(* CODESYS project T620X_HMI_CR1076_SP19p4.export

Project tree, tasks and I/O mapping:
  App_CODE_GEN/
    MAIN_CODE_GEN/
      App_CODE_GEN/
        Alarms/
          global variables GVL_Alarms
          program Alarms_Monitor_App [ST]
          program Alarms_Monitor_IO [ST]
        Diag_IO/
          program HMI_IO [FBD]: Init_Input_Links, Init_Output_Links, Update_Inputs, Update_Outputs
        Machine IO/
          Funcs/
            program Machine_Link_Inputs [ST]
            program Machine_Link_Inputs_Init [ST]
            program Machine_Link_Outputs [ST]
            program Machine_Link_Outputs_Init [ST]
            program Machine_Scale_Inputs [FBD]
          Structs/
            data type T620X_Radial_Inputs
            data type T620X_Radial_Outputs
    TEXT_LIST/
      text list AlarmGroup_App
      text list AlarmGroup_IO
      text list TextList_IO_Diag
*)

// App_CODE_GEN/MAIN_CODE_GEN/App_CODE_GEN/Machine IO/Structs/T620X_Radial_Inputs
TYPE T620X_Radial_Inputs :
STRUCT
// Machine_IO_Inputs_STRUCT_CODE_GEN_START

// generated (UTC): 2024-07-23 18:31:25.192393+00:00

ESTOP_OK:IpCom; // CHASSIS IN0100
DRUM_PRESSURE:IpCom; // CHASSIS IN0101
SPARE_IN0102:IpCom; // CHASSIS IN0102
SPARE_IN0103:IpCom; // CHASSIS IN0103
SPARE_IN0200:IpCom; // CHASSIS IN0200
SPARE_IN0201:IpCom; // CHASSIS IN0201
SPARE_IN0202:IpCom; // CHASSIS IN0202
SPARE_IN0203:IpCom; // CHASSIS IN0203
SPARE_IN0600:IpCom; // CHASSIS IN0600
SPARE_IN0601:IpCom; // CHASSIS IN0601
SPARE_IN0602:IpCom; // CHASSIS IN0602
SPARE_IN0603:IpCom; // CHASSIS IN0603
SPARE_IN0700:IpCom; // CHASSIS IN0700
RADIORHS_JACKLEGRAISE_REQ:IpCom; // CHASSIS IN0701
RHS_TROMMELDOORSW:IpCom; // CHASSIS IN0702
LHS_TROMMELDOORSW:IpCom; // CHASSIS IN0703
HYDOILTEMP_SW:IpCom; // CHASSIS IN0000
HYDOILLEVEL_SW:IpCom; // CHASSIS IN0001
THERMOSTAT:IpCom; // CHASSIS IN0002
RADIORHS_JACKLEGLOWER_REQ:IpCom; // CHASSIS IN0003
RADIOLHS_JACKLEGRAISE_REQ:IpCom; // CHASSIS IN0500
RADIOLHS_JACKLEGLOWER_REQ:IpCom; // CHASSIS IN0501
RADIOSIDECONVRAISEREQ:IpCom; // CHASSIS IN0502
RADIOSIDECONVLOWERREQ:IpCom; // CHASSIS IN0503
SPARE_IN0400:IpCom; // CHASSIS IN0400
FUELLEVEL_PERCENT:IpCom; // CHASSIS IN0401
UMBTRACKREQ:IpCom; // CHASSIS IN0900
UMBMACHINESTOP:IpCom; // CHASSIS IN0901
RTF_REQ:IpCom; // CHASSIS IN0300
RTR_REQ:IpCom; // CHASSIS IN0301
LTF_REQ:IpCom; // CHASSIS IN0800
LTR_REQ:IpCom; // CHASSIS IN0801


// Machine_IO_Inputs_STRUCT_CODE_GEN_STOP 

END_STRUCT
END_TYPE

// App_CODE_GEN/MAIN_CODE_GEN/App_CODE_GEN/Machine IO/Structs/T620X_Radial_Outputs
TYPE T620X_Radial_Outputs :
STRUCT
// Machine_IO_Outputs_STRUCT_CODE_GEN_START

// generated (UTC): 2024-07-23 18:31:25.208393+00:00

TAILCONVSPD_MA:OpCom; // CHASSIS.OUT0000
RHS_JACKLEGLOWER_OP:OpCom; // CHASSIS.OUT0001
SIDECONVSPD_MA:OpCom; // CHASSIS.OUT0002
LHS_JACKLEGRAISE_OP:OpCom; // CHASSIS.OUT0003
SIDETRANSFERSPD_MA:OpCom; // CHASSIS.OUT0004
LHS_JACKLEGLOWER_OP:OpCom; // CHASSIS.OUT0005
SETUPDUMPVALVE_OP:OpCom; // CHASSIS.OUT0006
COLLECTIONCONVSPD_MA:OpCom; // CHASSIS.OUT0007
COLLECTIONCONVON_OP:OpCom; // CHASSIS.OUT0008
SPARE_GROUP0:OpGrpCom; // CHASSIS.GROUP0
DRUMSPD_MA_RAMP_LIMIT:OpCom; // CHASSIS.OUT0100
TRACKINGMODE:OpCom; // CHASSIS.OUT0101
FEEDERSPD_MA:OpCom; // CHASSIS.OUT0102
CRANKENABLE:OpCom; // CHASSIS.OUT0103
DIVERTOILTOTRACK_OP:OpCom; // CHASSIS.OUT0104
RHS_JACKLEGRAISE_OP:OpCom; // CHASSIS.OUT0105
TAILCONVON_OP:OpCom; // CHASSIS.OUT0106
SIDECONVON_OP:OpCom; // CHASSIS.OUT0107
SIDETRANSFERON_OP:OpCom; // CHASSIS.OUT0108
SPARE_GROUP1:OpGrpCom; // CHASSIS.GROUP1
LEFTTRACKDIVERT_OP:OpCom; // CHASSIS.OUT0200
LTF_OP:OpCom; // CHASSIS.OUT0201
LTR_OP:OpCom; // CHASSIS.OUT0202
RIGHTTRACKDIVERT_OP:OpCom; // CHASSIS.OUT0203
RTF_OP:OpCom; // CHASSIS.OUT0204
RTR_OP:OpCom; // CHASSIS.OUT0205
DRUMONOFF_OP:OpCom; // CHASSIS.OUT0206
FEEDERONOFF_OP:OpCom; // CHASSIS.OUT0207
ECUENABLE:OpCom; // CHASSIS.OUT0208
SPARE_GROUP2:OpGrpCom; // CHASSIS.GROUP2
SPARE_OUT3000:OpCom; // CHASSIS.OUT3000
SPARE_OUT3001:OpCom; // CHASSIS.OUT3001


// Machine_IO_Outputs_STRUCT_CODE_GEN_STOP 	

END_STRUCT
END_TYPE

// App_CODE_GEN/MAIN_CODE_GEN/App_CODE_GEN/Alarms/GVL_Alarms
{attribute 'qualified_only'}
VAR_GLOBAL
// GVL_Alarms_Declare_CODE_GEN_START

// generated (UTC): 2024-07-23 18:31:25.263396+00:00

	EMERGENCY_STOP_COMMON: BOOL; // ID=101
	ETHERNET_PLC_COMMON_FAILURE: BOOL; // ID=102
	ETHERNET_CHASSIS_PLC_MISSING: BOOL; // ID=104
	ETHERNET_CHASSIS_PLC_ERROR_LT: BOOL; // ID=106
	ETHERNET_CHASSIS_PLC_ERROR_DIFF: BOOL; // ID=108
	ETHERNET_CHASSIS_PLC_ERROR_FROZEN: BOOL; // ID=110
	ETHERNET_CHASSIS_PLC_WARNING_DIFF: BOOL; // ID=112
	ETHERNET_CHASSIS_PLC_WARNING_FROZEN: BOOL; // ID=114
	Battery_Voltage_Warning: BOOL; // ID=118
	Hydraulic_Oil_Level_Low: BOOL; // ID=119
// GVL_Alarms_Declare_CODE_GEN_STOP
END_VAR

// App_CODE_GEN/MAIN_CODE_GEN/App_CODE_GEN/Alarms/Alarms_Monitor_App
PROGRAM Alarms_Monitor_App
VAR_INPUT
	LIST: REFERENCE TO SLL_LOGGER_MAIN_SRUCT;	
END_VAR
VAR
	App_Error_Group: SLL_LOGGER_ITEM_GROUP:=(ErrorApp:=1);	
	
// Alarms_Monitor_App_Declare_CODE_GEN_START

// generated (UTC): 2024-07-23 18:31:25.274396+00:00

	EMERGENCY_STOP_COMMON: SLL_AlarmBit;
	ETHERNET_PLC_COMMON_FAILURE: SLL_AlarmBit;
	ETHERNET_CHASSIS_PLC_MISSING: SLL_AlarmBit;
	ETHERNET_CHASSIS_PLC_ERROR_LT: SLL_AlarmBit;
	ETHERNET_CHASSIS_PLC_ERROR_DIFF: SLL_AlarmBit;
	ETHERNET_CHASSIS_PLC_ERROR_FROZEN: SLL_AlarmBit;
	ETHERNET_CHASSIS_PLC_WARNING_DIFF: SLL_AlarmBit;
	ETHERNET_CHASSIS_PLC_WARNING_FROZEN: SLL_AlarmBit;
	Battery_Voltage_Warning: SLL_AlarmBit;
	Hydraulic_Oil_Level_Low: SLL_AlarmBit;
	// Alarms_Monitor_App_Declare_CODE_GEN_STOP	
END_VAR


// Alarms_Monitor_App_STL_Body_CODE_GEN_START

// generated (UTC): 2024-07-23 18:31:25.284397+00:00

EMERGENCY_STOP_COMMON(LIST:=LIST,Bit_Input:=GVL_Alarms.EMERGENCY_STOP_COMMON,ID:=101,Add_Info:='',Group:=App_Error_Group,HushOption:=1);
ETHERNET_PLC_COMMON_FAILURE(LIST:=LIST,Bit_Input:=GVL_Alarms.ETHERNET_PLC_COMMON_FAILURE,ID:=102,Add_Info:='',Group:=App_Error_Group,HushOption:=0);
Battery_Voltage_Warning(LIST:=LIST,Bit_Input:=GVL_Alarms.Battery_Voltage_Warning,ID:=103,Add_Info:='',Group:=App_Error_Group,HushOption:=0);
Hydraulic_Oil_Level_Low(LIST:=LIST,Bit_Input:=GVL_Alarms.Hydraulic_Oil_Level_Low,ID:=104,Add_Info:='',Group:=App_Error_Group,HushOption:=0);

ETHERNET_CHASSIS_PLC_MISSING(LIST:=LIST,Bit_Input:=GVL_Alarms.ETHERNET_CHASSIS_PLC_MISSING,ID:=1100,Add_Info:='',Group:=App_Error_Group,HushOption:=0);
ETHERNET_CHASSIS_PLC_ERROR_LT(LIST:=LIST,Bit_Input:=GVL_Alarms.ETHERNET_CHASSIS_PLC_ERROR_LT,ID:=1101,Add_Info:='',Group:=App_Error_Group,HushOption:=0);
ETHERNET_CHASSIS_PLC_ERROR_DIFF(LIST:=LIST,Bit_Input:=GVL_Alarms.ETHERNET_CHASSIS_PLC_ERROR_DIFF,ID:=1102,Add_Info:='',Group:=App_Error_Group,HushOption:=0);
ETHERNET_CHASSIS_PLC_ERROR_FROZEN(LIST:=LIST,Bit_Input:=GVL_Alarms.ETHERNET_CHASSIS_PLC_ERROR_FROZEN,ID:=1103,Add_Info:='',Group:=App_Error_Group,HushOption:=0);
ETHERNET_CHASSIS_PLC_WARNING_DIFF(LIST:=LIST,Bit_Input:=GVL_Alarms.ETHERNET_CHASSIS_PLC_WARNING_DIFF,ID:=1104,Add_Info:='',Group:=App_Error_Group,HushOption:=0);
ETHERNET_CHASSIS_PLC_WARNING_FROZEN(LIST:=LIST,Bit_Input:=GVL_Alarms.ETHERNET_CHASSIS_PLC_WARNING_FROZEN,ID:=1105,Add_Info:='',Group:=App_Error_Group,HushOption:=0);




// Alarms_Monitor_App_STL_Body_CODE_GEN_STOP

END_PROGRAM

// App_CODE_GEN/MAIN_CODE_GEN/App_CODE_GEN/Alarms/Alarms_Monitor_IO
PROGRAM Alarms_Monitor_IO
VAR_INPUT
	LIST: REFERENCE TO SLL_LOGGER_MAIN_SRUCT;	
END_VAR
VAR
	IO_Error_Group: SLL_LOGGER_ITEM_GROUP:=(ErrorIO:=1);

// Alarms_Monitor_IO_Declare_CODE_GEN_START

// generated (UTC): 2024-07-23 18:31:25.297397+00:00

	ESTOPS_SAFETY_RELAY: SLL_AlarmBit;
	OVERRIDE_GENERAL_SWT: SLL_AlarmBit;
	FUNCTIONS_DEADMAN_CHASSIS_BTN: SLL_AlarmBit;
	CABIN_RAISE_CHASSIS_BTN: SLL_AlarmBit;
	CABIN_LOWER_CHASSIS_BTN: SLL_AlarmBit;
	JACKLEGS_DOWN_CHASSIS_BTN: SLL_AlarmBit;
	JACKLEGS_UP_CHASSIS_BTN: SLL_AlarmBit;
	ENGINE_START_CHASSIS_BTN: SLL_AlarmBit;
	HYDRAULICS_DC_PUMP_RUNNING_SIG: SLL_AlarmBit;
	JACKLEGS_STOWED_DOWN_PRESSURE_SWT: SLL_AlarmBit;
	JACKLEGS_STOWED_UP_PRESSURE_SWT: SLL_AlarmBit;
	MAINS_AC_MAINS_CONNECTED: SLL_AlarmBit;
	TRUCK_NEUTRAL_FROM_TRUCK : SLL_AlarmBit;
	SPARE_CHASSIS_IN0701: SLL_AlarmBit;
	CABIN_PART_RAISED_DIG: SLL_AlarmBit;
	SPARE_CHASSIS_IN0703: SLL_AlarmBit;
	CABIN_LOWER_LIMIT_DIG: SLL_AlarmBit;
	CABIN_FULLY_STOWED_DIG: SLL_AlarmBit;
	PTO_ACTIVE_SIG: SLL_AlarmBit;
	FUNCTIONS_CHASSIS_CABIN_CHANGE_OVER_SWT: SLL_AlarmBit;
	LIGHTS_SIDE_LIGHTS_DASH_SIG: SLL_AlarmBit;
	TRUCK_HANDBRAKE_APPLIED_SIGNAL: SLL_AlarmBit;
	ENGINE_RUNNING_SIGNAL: SLL_AlarmBit;
	TRUCK_REVERSE_FROM_TRUCK: SLL_AlarmBit;
	SPARE_CHASSIS_IN0400: SLL_AlarmBit;
	ENGINE_STOP_CHASSIS_BTN: SLL_AlarmBit;
	HYDRAULICS_OIL_LEVEL_RES: SLL_AlarmBit;
	SPARE_CHASSIS_IN0901: SLL_AlarmBit;
	SPARE_CHASSIS_IN0300: SLL_AlarmBit;
	SPARE_CHASSIS_IN0301: SLL_AlarmBit;
	JACKLEGS_CYCLINDER_100_BAR_PRESSURE_SWT: SLL_AlarmBit;
	JACKLEGS_CYCLINDER_150_BAR_PRESSURE_SWT: SLL_AlarmBit;
	ENGINE_STOP_COMMAND: SLL_AlarmBit;
	CHASSIS_SIREN: SLL_AlarmBit;
	SPARE_CHASSIS_OUT0002: SLL_AlarmBit;
	JACKLEGS_WARNING_BEACON: SLL_AlarmBit;
	HYDRAULICS_OIL_LEVEL_WARNING_LED: SLL_AlarmBit;
	SPARE_CHASSIS_OUT0005: SLL_AlarmBit;
	HYDRAULICS_MASTER_VALVE: SLL_AlarmBit;
	PTO_TOGGLE: SLL_AlarmBit;
	SPARE_CHASSIS_OUT0008: SLL_AlarmBit;
	CHASSIS_Supply_GROUP0: SLL_AlarmBit;
	SPARE_CHASSIS_OUT0100: SLL_AlarmBit;
	ENGINE_START_COMMAND: SLL_AlarmBit;
	SPARE_CHASSIS_OUT0102: SLL_AlarmBit;
	PLATFORM_TRAVERSE_LEFT_VALVE: SLL_AlarmBit;
	SPARE_CHASSIS_OUT0104: SLL_AlarmBit;
	CABIN_RAISE_COMMAND: SLL_AlarmBit;
	CABIN_LOWER_COMMAND: SLL_AlarmBit;
	JACKLEGS_UP_COMMAND: SLL_AlarmBit;
	JACKLEGS_DOWN_COMMAND: SLL_AlarmBit;
	CHASSIS_Supply_GROUP1: SLL_AlarmBit;
	HYDRAULICS_MASTER_LED_CAB: SLL_AlarmBit;
	OVERRIDE_DRIVE_INTERLOCK_ACTIVE_LED: SLL_AlarmBit;
	CABIN_FULLY_STOWED_LED: SLL_AlarmBit;
	JACKLEGS_STOWED_LED: SLL_AlarmBit;
	JACKLEGS_DOWN_LED: SLL_AlarmBit;
	CABIN_RAISED_LED: SLL_AlarmBit;
	PLATFORM_TRAVERSE_RIGHT_VALVE: SLL_AlarmBit;
	PLATFORM_RETRACT_COMMAND: SLL_AlarmBit;
	PLATFORM_EXTEND_COMMAND: SLL_AlarmBit;
	CHASSIS_Supply_GROUP2: SLL_AlarmBit;
	SPARE_CHASSIS_OUT3000: SLL_AlarmBit;
	SPARE_CHASSIS_OUT3001: SLL_AlarmBit;
	SPARE_CABIN_IN0100: SLL_AlarmBit;
	PLATFORM_EXTEND_BTN: SLL_AlarmBit;
	PLATFORM_RETRACT_BTN: SLL_AlarmBit;
	PLATFORM_SIDERAILS_LHS_SIDERAILS_STOWED_DIG: SLL_AlarmBit;
	PLATFORM_SIDERAILS_RHS_SIDERAILS_STOWED_DIG: SLL_AlarmBit;
	PLATFORM_TRAVERSE_STOWED_DIG: SLL_AlarmBit;
	SPARE_CABIN_IN0202: SLL_AlarmBit;
	PLATFORM_LEUZE_SENSORS_LEFT_SENSOR_DIG: SLL_AlarmBit;
	PLATFORM_LEUZE_SENSORS_RIGHT_SENSOR_DIG: SLL_AlarmBit;
	PLATFORM_FULLY_STOWED_DIG: SLL_AlarmBit;
	PLATFORM_PART_STOWED_DIG: SLL_AlarmBit;
	DOORS_REAR_DOOR_CLOSED_SIG: SLL_AlarmBit;
	PLATFORM_SAFETY_GATES_LHS_EDGE_SENSOR: SLL_AlarmBit;
	SPARE_CABIN_IN0701: SLL_AlarmBit;
	SPARE_CABIN_IN0702: SLL_AlarmBit;
	PLATFORM_SAFETY_GATES_RHS_EDGE_SENSOR: SLL_AlarmBit;
	SPARE_CABIN_IN0000: SLL_AlarmBit;
	PLATFORM_SAFETY_GATES_LHS_GATE_CLOSED_SIGNAL: SLL_AlarmBit;
	PLATFORM_SAFETY_GATES_RHS_GATE_CLOSED_SIGNAL: SLL_AlarmBit;
	SPARE_CABIN_IN0003: SLL_AlarmBit;
	CAS_RESET_SWT: SLL_AlarmBit;
	CAS_TORTOISE_SWT: SLL_AlarmBit;
	CAS_ENABLE_ON_OFF_SWT: SLL_AlarmBit;
	SPARE_CABIN_IN0503: SLL_AlarmBit;
	PLATFORM_SAFETY_EDGE_SAFETY_BUMPER_RES_ANA: SLL_AlarmBit;
	SPARE_CABIN_IN0401: SLL_AlarmBit;
	PLATFORM_TRAVERSE_LEFT_BTN: SLL_AlarmBit;
	PLATFORM_TRAVERSE_RIGHT_BTN: SLL_AlarmBit;
	DOORS_SIDE_DOOR_CLOSED_SIG: SLL_AlarmBit;
	FUNCTIONS_DEADMAN_CABIN_BTN: SLL_AlarmBit;
	SPARE_CABIN_IN0800: SLL_AlarmBit;
	SPARE_CABIN_IN0801: SLL_AlarmBit;
	PLATFORM_SIDERAILS_SIDERAILS_STOWED_LED: SLL_AlarmBit;
	PLATFORM_SAFETY_GATES_UNLOCK_1: SLL_AlarmBit;
	TRUCK_FORCE_NEUTRAL: SLL_AlarmBit;
	PLATFORM_SAFETY_GATES_UNLOCK_2: SLL_AlarmBit;
	CAS_LOCKOUT_LED: SLL_AlarmBit;
	PLATFORM_EXTENDED_LED: SLL_AlarmBit;
	PLATFORM_RETRACTED_LED: SLL_AlarmBit;
	CAS_TORTOISE_MODE_LED: SLL_AlarmBit;
	CAS_DRIVERS_BUZZER: SLL_AlarmBit;
	CABIN_Supply_GROUP0: SLL_AlarmBit;
	DOORS_ALLOW_SIDE_DOOR: SLL_AlarmBit;
	DOORS_ALLOW_REAR_DOOR: SLL_AlarmBit;
	SPARE_CABIN_OUT0102: SLL_AlarmBit;
	SPARE_CABIN_OUT0103: SLL_AlarmBit;
	SPARE_CABIN_OUT0104: SLL_AlarmBit;
	SPARE_CABIN_OUT0105: SLL_AlarmBit;
	SPARE_CABIN_OUT0106: SLL_AlarmBit;
	SPARE_CABIN_OUT0107: SLL_AlarmBit;
	SPARE_CABIN_OUT0108: SLL_AlarmBit;
	CABIN_Supply_GROUP1: SLL_AlarmBit;
	SPARE_CABIN_OUT0200: SLL_AlarmBit;
	LIGHTS_LEFT_SIDE_LIGHTS: SLL_AlarmBit;
	CAS_GREEN_BEACON: SLL_AlarmBit;
	FUNCTIONS_DEADMAN_CABIN_BTN_LED: SLL_AlarmBit;
	SPARE_CABIN_OUT0204: SLL_AlarmBit;
	SPARE_CABIN_OUT0205: SLL_AlarmBit;
	LIGHTS_SIDE_RLY: SLL_AlarmBit;
	SPARE_CABIN_OUT0207: SLL_AlarmBit;
	SPARE_CABIN_OUT0208: SLL_AlarmBit;
	CABIN_Supply_GROUP2: SLL_AlarmBit;
	SPARE_CABIN_OUT3000: SLL_AlarmBit;
	SPARE_CABIN_OUT3001: SLL_AlarmBit;
	// Alarms_Monitor_IO_Declare_CODE_GEN_STOP	
END_VAR


// Alarms_Monitor_IO_STL_Body_CODE_GEN_START

// generated (UTC): 2024-07-23 18:31:25.307398+00:00

// Alarms_Monitor_IO_STL_Body_CODE_GEN_STOP

END_PROGRAM

// App_CODE_GEN/MAIN_CODE_GEN/App_CODE_GEN/Diag_IO/HMI_IO
PROGRAM HMI_IO
VAR
	Init_Link_Inputs: BOOL:=TRUE;
	Init_Link_Outputs: BOOL:=TRUE;
	CHASSIS: HMI_PLC_CR0709_IO;	
	Outputs_EnableAutoMan:BOOL:=TRUE;// AW TEMP 02-03-2024
	Wait_For_UDP_TON: TON;
END_VAR

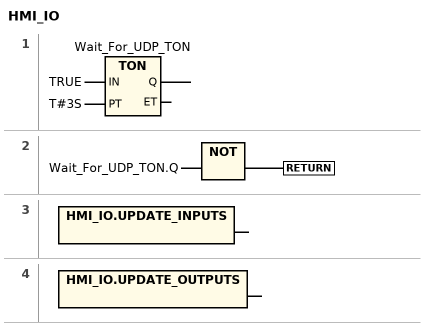
// NETWORK 1
Wait_For_UDP_TON(IN := TRUE, PT := T#3S); // TON

// NETWORK 2
IF NOT Wait_For_UDP_TON.Q THEN RETURN; END_IF

// NETWORK 3
HMI_IO.UPDATE_INPUTS();

// NETWORK 4
HMI_IO.UPDATE_OUTPUTS();

METHOD Init_Input_Links
VAR
END_VAR

// HMI_IO_Init_Input_Links_CODE_GEN_START

// generated (UTC): 2024-07-23 18:31:25.317398+00:00
CHASSIS.IN0100.Init(Machine_IO.Inputs.ESTOP_OK);
CHASSIS.IN0101.Init(Machine_IO.Inputs.DRUM_PRESSURE);
CHASSIS.IN0102.Init(Machine_IO.Inputs.SPARE_IN0102);
CHASSIS.IN0103.Init(Machine_IO.Inputs.SPARE_IN0103);
CHASSIS.IN0200.Init(Machine_IO.Inputs.SPARE_IN0200);
CHASSIS.IN0201.Init(Machine_IO.Inputs.SPARE_IN0201);
CHASSIS.IN0202.Init(Machine_IO.Inputs.SPARE_IN0202);
CHASSIS.IN0203.Init(Machine_IO.Inputs.SPARE_IN0203);
CHASSIS.IN0600.Init(Machine_IO.Inputs.SPARE_IN0600);
CHASSIS.IN0601.Init(Machine_IO.Inputs.SPARE_IN0601);
CHASSIS.IN0602.Init(Machine_IO.Inputs.SPARE_IN0602);
CHASSIS.IN0603.Init(Machine_IO.Inputs.SPARE_IN0603);
CHASSIS.IN0700.Init(Machine_IO.Inputs.SPARE_IN0700);
CHASSIS.IN0701.Init(Machine_IO.Inputs.RADIORHS_JACKLEGRAISE_REQ);
CHASSIS.IN0702.Init(Machine_IO.Inputs.RHS_TROMMELDOORSW);
CHASSIS.IN0703.Init(Machine_IO.Inputs.LHS_TROMMELDOORSW);
CHASSIS.IN0000.Init(Machine_IO.Inputs.HYDOILTEMP_SW);
CHASSIS.IN0001.Init(Machine_IO.Inputs.HYDOILLEVEL_SW);
CHASSIS.IN0002.Init(Machine_IO.Inputs.THERMOSTAT);
CHASSIS.IN0003.Init(Machine_IO.Inputs.RADIORHS_JACKLEGLOWER_REQ);
CHASSIS.IN0500.Init(Machine_IO.Inputs.RADIOLHS_JACKLEGRAISE_REQ);
CHASSIS.IN0501.Init(Machine_IO.Inputs.RADIOLHS_JACKLEGLOWER_REQ);
CHASSIS.IN0502.Init(Machine_IO.Inputs.RADIOSIDECONVRAISEREQ);
CHASSIS.IN0503.Init(Machine_IO.Inputs.RADIOSIDECONVLOWERREQ);
CHASSIS.IN0400.Init(Machine_IO.Inputs.SPARE_IN0400);
CHASSIS.IN0401.Init(Machine_IO.Inputs.FUELLEVEL_PERCENT);
CHASSIS.IN0900.Init(Machine_IO.Inputs.UMBTRACKREQ);
CHASSIS.IN0901.Init(Machine_IO.Inputs.UMBMACHINESTOP);
CHASSIS.IN0300.Init(Machine_IO.Inputs.RTF_REQ);
CHASSIS.IN0301.Init(Machine_IO.Inputs.RTR_REQ);
CHASSIS.IN0800.Init(Machine_IO.Inputs.LTF_REQ);
CHASSIS.IN0801.Init(Machine_IO.Inputs.LTR_REQ);

// HMI_IO_Init_Input_Links_CODE_GEN_STOP
END_METHOD

METHOD Init_Output_Links
VAR
END_VAR

// HMI_IO_Init_Output_Links_CODE_GEN_START

// generated (UTC): 2024-07-23 18:31:25.327399+00:00
CHASSIS.OUT0000.Init(Machine_IO.Outputs.TAILCONVSPD_MA);
CHASSIS.OUT0001.Init(Machine_IO.Outputs.RHS_JACKLEGLOWER_OP);
CHASSIS.OUT0002.Init(Machine_IO.Outputs.SIDECONVSPD_MA);
CHASSIS.OUT0003.Init(Machine_IO.Outputs.LHS_JACKLEGRAISE_OP);
CHASSIS.OUT0004.Init(Machine_IO.Outputs.SIDETRANSFERSPD_MA);
CHASSIS.OUT0005.Init(Machine_IO.Outputs.LHS_JACKLEGLOWER_OP);
CHASSIS.OUT0006.Init(Machine_IO.Outputs.SETUPDUMPVALVE_OP);
CHASSIS.OUT0007.Init(Machine_IO.Outputs.COLLECTIONCONVSPD_MA);
CHASSIS.OUT0008.Init(Machine_IO.Outputs.COLLECTIONCONVON_OP);
CHASSIS.GROUP0.Init(Machine_IO.Outputs.SPARE_GROUP0);
CHASSIS.OUT0100.Init(Machine_IO.Outputs.DRUMSPD_MA_RAMP_LIMIT);
CHASSIS.OUT0101.Init(Machine_IO.Outputs.TRACKINGMODE);
CHASSIS.OUT0102.Init(Machine_IO.Outputs.FEEDERSPD_MA);
CHASSIS.OUT0103.Init(Machine_IO.Outputs.CRANKENABLE);
CHASSIS.OUT0104.Init(Machine_IO.Outputs.DIVERTOILTOTRACK_OP);
CHASSIS.OUT0105.Init(Machine_IO.Outputs.RHS_JACKLEGRAISE_OP);
CHASSIS.OUT0106.Init(Machine_IO.Outputs.TAILCONVON_OP);
CHASSIS.OUT0107.Init(Machine_IO.Outputs.SIDECONVON_OP);
CHASSIS.OUT0108.Init(Machine_IO.Outputs.SIDETRANSFERON_OP);
CHASSIS.GROUP1.Init(Machine_IO.Outputs.SPARE_GROUP1);
CHASSIS.OUT0200.Init(Machine_IO.Outputs.LEFTTRACKDIVERT_OP);
CHASSIS.OUT0201.Init(Machine_IO.Outputs.LTF_OP);
CHASSIS.OUT0202.Init(Machine_IO.Outputs.LTR_OP);
CHASSIS.OUT0203.Init(Machine_IO.Outputs.RIGHTTRACKDIVERT_OP);
CHASSIS.OUT0204.Init(Machine_IO.Outputs.RTF_OP);
CHASSIS.OUT0205.Init(Machine_IO.Outputs.RTR_OP);
CHASSIS.OUT0206.Init(Machine_IO.Outputs.DRUMONOFF_OP);
CHASSIS.OUT0207.Init(Machine_IO.Outputs.FEEDERONOFF_OP);
CHASSIS.OUT0208.Init(Machine_IO.Outputs.ECUENABLE);
CHASSIS.GROUP2.Init(Machine_IO.Outputs.SPARE_GROUP2);
CHASSIS.OUT3000.Init(Machine_IO.Outputs.SPARE_OUT3000);
CHASSIS.OUT3001.Init(Machine_IO.Outputs.SPARE_OUT3001);

// HMI_IO_Init_Output_Links_CODE_GEN_STOP
END_METHOD

METHOD Update_Inputs
VAR	
END_VAR
IF Init_Link_Inputs THEN
	Init_Input_Links();
END_IF
Init_Link_Inputs:=FALSE;

// HMI_IO_Update_Inputs_CODE_GEN_START

// generated (UTC): 2024-07-23 18:31:25.338400+00:00

CHASSIS.IN0100();
CHASSIS.IN0101();
CHASSIS.IN0102();
CHASSIS.IN0103();
CHASSIS.IN0200();
CHASSIS.IN0201();
CHASSIS.IN0202();
CHASSIS.IN0203();
CHASSIS.IN0600();
CHASSIS.IN0601();
CHASSIS.IN0602();
CHASSIS.IN0603();
CHASSIS.IN0700();
CHASSIS.IN0701();
CHASSIS.IN0702();
CHASSIS.IN0703();
CHASSIS.IN0000();
CHASSIS.IN0001();
CHASSIS.IN0002();
CHASSIS.IN0003();
CHASSIS.IN0500();
CHASSIS.IN0501();
CHASSIS.IN0502();
CHASSIS.IN0503();
CHASSIS.IN0400();
CHASSIS.IN0401();
CHASSIS.IN0900();
CHASSIS.IN0901();
CHASSIS.IN0300();
CHASSIS.IN0301();
CHASSIS.IN0800();
CHASSIS.IN0801();
// HMI_IO_Update_Inputs_CODE_GEN_STOP
END_METHOD

METHOD Update_Outputs
VAR
END_VAR
IF Init_Link_Outputs THEN
	Init_Output_Links();
END_IF
Init_Link_Outputs:=FALSE;

// HMI_IO_Update_Outputs_CODE_GEN_START

// generated (UTC): 2024-07-23 18:31:25.349399+00:00

CHASSIS.OUT0000();
CHASSIS.OUT0001();
CHASSIS.OUT0002();
CHASSIS.OUT0003();
CHASSIS.OUT0004();
CHASSIS.OUT0005();
CHASSIS.OUT0006();
CHASSIS.OUT0007();
CHASSIS.OUT0008();
CHASSIS.GROUP0();
CHASSIS.OUT0100();
CHASSIS.OUT0101();
CHASSIS.OUT0102();
CHASSIS.OUT0103();
CHASSIS.OUT0104();
CHASSIS.OUT0105();
CHASSIS.OUT0106();
CHASSIS.OUT0107();
CHASSIS.OUT0108();
CHASSIS.GROUP1();
CHASSIS.OUT0200();
CHASSIS.OUT0201();
CHASSIS.OUT0202();
CHASSIS.OUT0203();
CHASSIS.OUT0204();
CHASSIS.OUT0205();
CHASSIS.OUT0206();
CHASSIS.OUT0207();
CHASSIS.OUT0208();
CHASSIS.GROUP2();
CHASSIS.OUT3000();
CHASSIS.OUT3001();
// HMI_IO_Update_Outputs_CODE_GEN_STOP
END_METHOD

END_PROGRAM

// App_CODE_GEN/MAIN_CODE_GEN/App_CODE_GEN/Machine IO/Funcs/Machine_Link_Inputs
PROGRAM Machine_Link_Inputs
VAR_INPUT
	ENA:BOOL;
END_VAR

VAR
	INIT_ONCE:BOOL:=TRUE;
	Init_Input_Links:BOOL :=TRUE;
END_VAR

IF Init_Input_Links THEN
	Machine_Link_Inputs_Init();	
	Init_Input_Links:=FALSE;
END_IF

// Machine_Link_Inputs_Main_CODE_GEN_START

// generated (UTC): 2024-07-23 18:31:25.048386+00:00

Machine_IO.Inputs.ESTOP_OK(); // CR0709.IN0100
Machine_IO.Inputs.DRUM_PRESSURE(); // CR0709.IN0101
Machine_IO.Inputs.SPARE_IN0102(); // CR0709.IN0102
Machine_IO.Inputs.SPARE_IN0103(); // CR0709.IN0103
Machine_IO.Inputs.SPARE_IN0200(); // CR0709.IN0200
Machine_IO.Inputs.SPARE_IN0201(); // CR0709.IN0201
Machine_IO.Inputs.SPARE_IN0202(); // CR0709.IN0202
Machine_IO.Inputs.SPARE_IN0203(); // CR0709.IN0203
Machine_IO.Inputs.SPARE_IN0600(); // CR0709.IN0600
Machine_IO.Inputs.SPARE_IN0601(); // CR0709.IN0601
Machine_IO.Inputs.SPARE_IN0602(); // CR0709.IN0602
Machine_IO.Inputs.SPARE_IN0603(); // CR0709.IN0603
Machine_IO.Inputs.SPARE_IN0700(); // CR0709.IN0700
Machine_IO.Inputs.RADIORHS_JACKLEGRAISE_REQ(); // CR0709.IN0701
Machine_IO.Inputs.RHS_TROMMELDOORSW(); // CR0709.IN0702
Machine_IO.Inputs.LHS_TROMMELDOORSW(); // CR0709.IN0703
Machine_IO.Inputs.HYDOILTEMP_SW(); // CR0709.IN0000
Machine_IO.Inputs.HYDOILLEVEL_SW(); // CR0709.IN0001
Machine_IO.Inputs.THERMOSTAT(); // CR0709.IN0002
Machine_IO.Inputs.RADIORHS_JACKLEGLOWER_REQ(); // CR0709.IN0003
Machine_IO.Inputs.RADIOLHS_JACKLEGRAISE_REQ(); // CR0709.IN0500
Machine_IO.Inputs.RADIOLHS_JACKLEGLOWER_REQ(); // CR0709.IN0501
Machine_IO.Inputs.RADIOSIDECONVRAISEREQ(); // CR0709.IN0502
Machine_IO.Inputs.RADIOSIDECONVLOWERREQ(); // CR0709.IN0503
Machine_IO.Inputs.SPARE_IN0400(); // CR0709.IN0400
Machine_IO.Inputs.FUELLEVEL_PERCENT(); // CR0709.IN0401
Machine_IO.Inputs.UMBTRACKREQ(); // CR0709.IN0900
Machine_IO.Inputs.UMBMACHINESTOP(); // CR0709.IN0901
Machine_IO.Inputs.RTF_REQ(); // CR0709.IN0300
Machine_IO.Inputs.RTR_REQ(); // CR0709.IN0301
Machine_IO.Inputs.LTF_REQ(); // CR0709.IN0800
Machine_IO.Inputs.LTR_REQ(); // CR0709.IN0801


// Machine_Link_Inputs_Main_CODE_GEN_STOP

END_PROGRAM

// App_CODE_GEN/MAIN_CODE_GEN/App_CODE_GEN/Machine IO/Funcs/Machine_Link_Inputs_Init
PROGRAM Machine_Link_Inputs_Init
VAR
END_VAR


// Machine_Link_Inputs_Init_CODE_GEN_START

// generated (UTC): 2024-07-23 18:31:25.086388+00:00
Machine_IO.Inputs.ESTOP_OK.Init('CHASSIS','ESTOP_OK','IN0100','a63',NVL_IO_CHASSIS.All_Inputs.IN0100,Machine_IO.Node_CHASSIS);
Machine_IO.Inputs.DRUM_PRESSURE.Init('CHASSIS','DRUM_PRESSURE','IN0101','a64',NVL_IO_CHASSIS.All_Inputs.IN0101,Machine_IO.Node_CHASSIS);
Machine_IO.Inputs.SPARE_IN0102.Init('CHASSIS','SPARE_IN0102','IN0102','a65',NVL_IO_CHASSIS.All_Inputs.IN0102,Machine_IO.Node_CHASSIS);
Machine_IO.Inputs.SPARE_IN0103.Init('CHASSIS','SPARE_IN0103','IN0103','a66',NVL_IO_CHASSIS.All_Inputs.IN0103,Machine_IO.Node_CHASSIS);
Machine_IO.Inputs.SPARE_IN0200.Init('CHASSIS','SPARE_IN0200','IN0200','a67',NVL_IO_CHASSIS.All_Inputs.IN0200,Machine_IO.Node_CHASSIS);
Machine_IO.Inputs.SPARE_IN0201.Init('CHASSIS','SPARE_IN0201','IN0201','a68',NVL_IO_CHASSIS.All_Inputs.IN0201,Machine_IO.Node_CHASSIS);
Machine_IO.Inputs.SPARE_IN0202.Init('CHASSIS','SPARE_IN0202','IN0202','a69',NVL_IO_CHASSIS.All_Inputs.IN0202,Machine_IO.Node_CHASSIS);
Machine_IO.Inputs.SPARE_IN0203.Init('CHASSIS','SPARE_IN0203','IN0203','a70',NVL_IO_CHASSIS.All_Inputs.IN0203,Machine_IO.Node_CHASSIS);
Machine_IO.Inputs.SPARE_IN0600.Init('CHASSIS','SPARE_IN0600','IN0600','a55',NVL_IO_CHASSIS.All_Inputs.IN0600,Machine_IO.Node_CHASSIS);
Machine_IO.Inputs.SPARE_IN0601.Init('CHASSIS','SPARE_IN0601','IN0601','a56',NVL_IO_CHASSIS.All_Inputs.IN0601,Machine_IO.Node_CHASSIS);
Machine_IO.Inputs.SPARE_IN0602.Init('CHASSIS','SPARE_IN0602','IN0602','a57',NVL_IO_CHASSIS.All_Inputs.IN0602,Machine_IO.Node_CHASSIS);
Machine_IO.Inputs.SPARE_IN0603.Init('CHASSIS','SPARE_IN0603','IN0603','a58',NVL_IO_CHASSIS.All_Inputs.IN0603,Machine_IO.Node_CHASSIS);
Machine_IO.Inputs.SPARE_IN0700.Init('CHASSIS','SPARE_IN0700','IN0700','a59',NVL_IO_CHASSIS.All_Inputs.IN0700,Machine_IO.Node_CHASSIS);
Machine_IO.Inputs.RADIORHS_JACKLEGRAISE_REQ.Init('CHASSIS','RADIORHS_JACKLEGRAISE_REQ','IN0701','a60',NVL_IO_CHASSIS.All_Inputs.IN0701,Machine_IO.Node_CHASSIS);
Machine_IO.Inputs.RHS_TROMMELDOORSW.Init('CHASSIS','RHS_TROMMELDOORSW','IN0702','a61',NVL_IO_CHASSIS.All_Inputs.IN0702,Machine_IO.Node_CHASSIS);
Machine_IO.Inputs.LHS_TROMMELDOORSW.Init('CHASSIS','LHS_TROMMELDOORSW','IN0703','a62',NVL_IO_CHASSIS.All_Inputs.IN0703,Machine_IO.Node_CHASSIS);
Machine_IO.Inputs.HYDOILTEMP_SW.Init('CHASSIS','HYDOILTEMP_SW','IN0000','a25',NVL_IO_CHASSIS.All_Inputs.IN0000,Machine_IO.Node_CHASSIS);
Machine_IO.Inputs.HYDOILLEVEL_SW.Init('CHASSIS','HYDOILLEVEL_SW','IN0001','a26',NVL_IO_CHASSIS.All_Inputs.IN0001,Machine_IO.Node_CHASSIS);
Machine_IO.Inputs.THERMOSTAT.Init('CHASSIS','THERMOSTAT','IN0002','a27',NVL_IO_CHASSIS.All_Inputs.IN0002,Machine_IO.Node_CHASSIS);
Machine_IO.Inputs.RADIORHS_JACKLEGLOWER_REQ.Init('CHASSIS','RADIORHS_JACKLEGLOWER_REQ','IN0003','a28',NVL_IO_CHASSIS.All_Inputs.IN0003,Machine_IO.Node_CHASSIS);
Machine_IO.Inputs.RADIOLHS_JACKLEGRAISE_REQ.Init('CHASSIS','RADIOLHS_JACKLEGRAISE_REQ','IN0500','a40',NVL_IO_CHASSIS.All_Inputs.IN0500,Machine_IO.Node_CHASSIS);
Machine_IO.Inputs.RADIOLHS_JACKLEGLOWER_REQ.Init('CHASSIS','RADIOLHS_JACKLEGLOWER_REQ','IN0501','a41',NVL_IO_CHASSIS.All_Inputs.IN0501,Machine_IO.Node_CHASSIS);
Machine_IO.Inputs.RADIOSIDECONVRAISEREQ.Init('CHASSIS','RADIOSIDECONVRAISEREQ','IN0502','a42',NVL_IO_CHASSIS.All_Inputs.IN0502,Machine_IO.Node_CHASSIS);
Machine_IO.Inputs.RADIOSIDECONVLOWERREQ.Init('CHASSIS','RADIOSIDECONVLOWERREQ','IN0503','a43',NVL_IO_CHASSIS.All_Inputs.IN0503,Machine_IO.Node_CHASSIS);
Machine_IO.Inputs.SPARE_IN0400.Init('CHASSIS','SPARE_IN0400','IN0400','a46',NVL_IO_CHASSIS.All_Inputs.IN0400,Machine_IO.Node_CHASSIS);
Machine_IO.Inputs.FUELLEVEL_PERCENT.Init('CHASSIS','FUELLEVEL_PERCENT','IN0401','a47',NVL_IO_CHASSIS.All_Inputs.IN0401,Machine_IO.Node_CHASSIS);
Machine_IO.Inputs.UMBTRACKREQ.Init('CHASSIS','UMBTRACKREQ','IN0900','a38',NVL_IO_CHASSIS.All_Inputs.IN0900,Machine_IO.Node_CHASSIS);
Machine_IO.Inputs.UMBMACHINESTOP.Init('CHASSIS','UMBMACHINESTOP','IN0901','a39',NVL_IO_CHASSIS.All_Inputs.IN0901,Machine_IO.Node_CHASSIS);
Machine_IO.Inputs.RTF_REQ.Init('CHASSIS','RTF_REQ','IN0300','a44',NVL_IO_CHASSIS.All_Inputs.IN0300,Machine_IO.Node_CHASSIS);
Machine_IO.Inputs.RTR_REQ.Init('CHASSIS','RTR_REQ','IN0301','a45',NVL_IO_CHASSIS.All_Inputs.IN0301,Machine_IO.Node_CHASSIS);
Machine_IO.Inputs.LTF_REQ.Init('CHASSIS','LTF_REQ','IN0800','a36',NVL_IO_CHASSIS.All_Inputs.IN0800,Machine_IO.Node_CHASSIS);
Machine_IO.Inputs.LTR_REQ.Init('CHASSIS','LTR_REQ','IN0801','a37',NVL_IO_CHASSIS.All_Inputs.IN0801,Machine_IO.Node_CHASSIS);


// Machine_Link_Inputs_Init_CODE_GEN_STOP

END_PROGRAM

// App_CODE_GEN/MAIN_CODE_GEN/App_CODE_GEN/Machine IO/Funcs/Machine_Link_Outputs
PROGRAM Machine_Link_Outputs
VAR_INPUT
	ENA:BOOL;
END_VAR
VAR
	Init_Output_Links: BOOL := TRUE;
END_VAR

IF ENA = FALSE THEN
	RETURN;
END_IF

IF Init_Output_Links THEN
	Machine_Link_Outputs_Init();
	Init_Output_Links:=FALSE;
END_IF

// Machine_Link_Outputs_Main_CODE_GEN_START

// generated (UTC): 2024-07-23 18:31:25.127390+00:00
Machine_IO.Outputs.TAILCONVSPD_MA(); // CR0709.OUT0000
Machine_IO.Outputs.RHS_JACKLEGLOWER_OP(); // CR0709.OUT0001
Machine_IO.Outputs.SIDECONVSPD_MA(); // CR0709.OUT0002
Machine_IO.Outputs.LHS_JACKLEGRAISE_OP(); // CR0709.OUT0003
Machine_IO.Outputs.SIDETRANSFERSPD_MA(); // CR0709.OUT0004
Machine_IO.Outputs.LHS_JACKLEGLOWER_OP(); // CR0709.OUT0005
Machine_IO.Outputs.SETUPDUMPVALVE_OP(); // CR0709.OUT0006
Machine_IO.Outputs.COLLECTIONCONVSPD_MA(); // CR0709.OUT0007
Machine_IO.Outputs.COLLECTIONCONVON_OP(); // CR0709.OUT0008
Machine_IO.Outputs.SPARE_GROUP0(); // CR0709.GROUP0
Machine_IO.Outputs.DRUMSPD_MA_RAMP_LIMIT(); // CR0709.OUT0100
Machine_IO.Outputs.TRACKINGMODE(); // CR0709.OUT0101
Machine_IO.Outputs.FEEDERSPD_MA(); // CR0709.OUT0102
Machine_IO.Outputs.CRANKENABLE(); // CR0709.OUT0103
Machine_IO.Outputs.DIVERTOILTOTRACK_OP(); // CR0709.OUT0104
Machine_IO.Outputs.RHS_JACKLEGRAISE_OP(); // CR0709.OUT0105
Machine_IO.Outputs.TAILCONVON_OP(); // CR0709.OUT0106
Machine_IO.Outputs.SIDECONVON_OP(); // CR0709.OUT0107
Machine_IO.Outputs.SIDETRANSFERON_OP(); // CR0709.OUT0108
Machine_IO.Outputs.SPARE_GROUP1(); // CR0709.GROUP1
Machine_IO.Outputs.LEFTTRACKDIVERT_OP(); // CR0709.OUT0200
Machine_IO.Outputs.LTF_OP(); // CR0709.OUT0201
Machine_IO.Outputs.LTR_OP(); // CR0709.OUT0202
Machine_IO.Outputs.RIGHTTRACKDIVERT_OP(); // CR0709.OUT0203
Machine_IO.Outputs.RTF_OP(); // CR0709.OUT0204
Machine_IO.Outputs.RTR_OP(); // CR0709.OUT0205
Machine_IO.Outputs.DRUMONOFF_OP(); // CR0709.OUT0206
Machine_IO.Outputs.FEEDERONOFF_OP(); // CR0709.OUT0207
Machine_IO.Outputs.ECUENABLE(); // CR0709.OUT0208
Machine_IO.Outputs.SPARE_GROUP2(); // CR0709.GROUP2
Machine_IO.Outputs.SPARE_OUT3000(); // CR0709.OUT3000
Machine_IO.Outputs.SPARE_OUT3001(); // CR0709.OUT3001

// Machine_Link_Outputs_Main_CODE_GEN_STOP

END_PROGRAM

// App_CODE_GEN/MAIN_CODE_GEN/App_CODE_GEN/Machine IO/Funcs/Machine_Link_Outputs_Init
PROGRAM Machine_Link_Outputs_Init
VAR
END_VAR


// Machine_Link_Outputs_Init_CODE_GEN_START

// generated (UTC): 2024-07-23 18:31:25.139390+00:00

Machine_IO.Outputs.TAILCONVSPD_MA.Init('CHASSIS','TAILCONVSPD_MA','OUT0000','a16',NVL_Outputs_States_CHASSIS.All.OUT0000,NVL_IO_CHASSIS.All_Outputs_Diag.OUT0000,Machine_IO.Node_CHASSIS);
Machine_IO.Outputs.RHS_JACKLEGLOWER_OP.Init('CHASSIS','RHS_JACKLEGLOWER_OP','OUT0001','a17',NVL_Outputs_States_CHASSIS.All.OUT0001,NVL_IO_CHASSIS.All_Outputs_Diag.OUT0001,Machine_IO.Node_CHASSIS);
Machine_IO.Outputs.SIDECONVSPD_MA.Init('CHASSIS','SIDECONVSPD_MA','OUT0002','a18',NVL_Outputs_States_CHASSIS.All.OUT0002,NVL_IO_CHASSIS.All_Outputs_Diag.OUT0002,Machine_IO.Node_CHASSIS);
Machine_IO.Outputs.LHS_JACKLEGRAISE_OP.Init('CHASSIS','LHS_JACKLEGRAISE_OP','OUT0003','a19',NVL_Outputs_States_CHASSIS.All.OUT0003,NVL_IO_CHASSIS.All_Outputs_Diag.OUT0003,Machine_IO.Node_CHASSIS);
Machine_IO.Outputs.SIDETRANSFERSPD_MA.Init('CHASSIS','SIDETRANSFERSPD_MA','OUT0004','a20',NVL_Outputs_States_CHASSIS.All.OUT0004,NVL_IO_CHASSIS.All_Outputs_Diag.OUT0004,Machine_IO.Node_CHASSIS);
Machine_IO.Outputs.LHS_JACKLEGLOWER_OP.Init('CHASSIS','LHS_JACKLEGLOWER_OP','OUT0005','a21',NVL_Outputs_States_CHASSIS.All.OUT0005,NVL_IO_CHASSIS.All_Outputs_Diag.OUT0005,Machine_IO.Node_CHASSIS);
Machine_IO.Outputs.SETUPDUMPVALVE_OP.Init('CHASSIS','SETUPDUMPVALVE_OP','OUT0006','a22',NVL_Outputs_States_CHASSIS.All.OUT0006,NVL_IO_CHASSIS.All_Outputs_Diag.OUT0006,Machine_IO.Node_CHASSIS);
Machine_IO.Outputs.COLLECTIONCONVSPD_MA.Init('CHASSIS','COLLECTIONCONVSPD_MA','OUT0007','a23',NVL_Outputs_States_CHASSIS.All.OUT0007,NVL_IO_CHASSIS.All_Outputs_Diag.OUT0007,Machine_IO.Node_CHASSIS);
Machine_IO.Outputs.COLLECTIONCONVON_OP.Init('CHASSIS','COLLECTIONCONVON_OP','OUT0008','a24',NVL_Outputs_States_CHASSIS.All.OUT0008,NVL_IO_CHASSIS.All_Outputs_Diag.OUT0008,Machine_IO.Node_CHASSIS);
Machine_IO.Outputs.DRUMSPD_MA_RAMP_LIMIT.Init('CHASSIS','DRUMSPD_MA_RAMP_LIMIT','OUT0100','a6',NVL_Outputs_States_CHASSIS.All.OUT0100,NVL_IO_CHASSIS.All_Outputs_Diag.OUT0100,Machine_IO.Node_CHASSIS);
Machine_IO.Outputs.TRACKINGMODE.Init('CHASSIS','TRACKINGMODE','OUT0101','a7',NVL_Outputs_States_CHASSIS.All.OUT0101,NVL_IO_CHASSIS.All_Outputs_Diag.OUT0101,Machine_IO.Node_CHASSIS);
Machine_IO.Outputs.FEEDERSPD_MA.Init('CHASSIS','FEEDERSPD_MA','OUT0102','a8',NVL_Outputs_States_CHASSIS.All.OUT0102,NVL_IO_CHASSIS.All_Outputs_Diag.OUT0102,Machine_IO.Node_CHASSIS);
Machine_IO.Outputs.CRANKENABLE.Init('CHASSIS','CRANKENABLE','OUT0103','a9',NVL_Outputs_States_CHASSIS.All.OUT0103,NVL_IO_CHASSIS.All_Outputs_Diag.OUT0103,Machine_IO.Node_CHASSIS);
Machine_IO.Outputs.DIVERTOILTOTRACK_OP.Init('CHASSIS','DIVERTOILTOTRACK_OP','OUT0104','a10',NVL_Outputs_States_CHASSIS.All.OUT0104,NVL_IO_CHASSIS.All_Outputs_Diag.OUT0104,Machine_IO.Node_CHASSIS);
Machine_IO.Outputs.RHS_JACKLEGRAISE_OP.Init('CHASSIS','RHS_JACKLEGRAISE_OP','OUT0105','a11',NVL_Outputs_States_CHASSIS.All.OUT0105,NVL_IO_CHASSIS.All_Outputs_Diag.OUT0105,Machine_IO.Node_CHASSIS);
Machine_IO.Outputs.TAILCONVON_OP.Init('CHASSIS','TAILCONVON_OP','OUT0106','a12',NVL_Outputs_States_CHASSIS.All.OUT0106,NVL_IO_CHASSIS.All_Outputs_Diag.OUT0106,Machine_IO.Node_CHASSIS);
Machine_IO.Outputs.SIDECONVON_OP.Init('CHASSIS','SIDECONVON_OP','OUT0107','a13',NVL_Outputs_States_CHASSIS.All.OUT0107,NVL_IO_CHASSIS.All_Outputs_Diag.OUT0107,Machine_IO.Node_CHASSIS);
Machine_IO.Outputs.SIDETRANSFERON_OP.Init('CHASSIS','SIDETRANSFERON_OP','OUT0108','a14',NVL_Outputs_States_CHASSIS.All.OUT0108,NVL_IO_CHASSIS.All_Outputs_Diag.OUT0108,Machine_IO.Node_CHASSIS);
Machine_IO.Outputs.LEFTTRACKDIVERT_OP.Init('CHASSIS','LEFTTRACKDIVERT_OP','OUT0200','a73',NVL_Outputs_States_CHASSIS.All.OUT0200,NVL_IO_CHASSIS.All_Outputs_Diag.OUT0200,Machine_IO.Node_CHASSIS);
Machine_IO.Outputs.LTF_OP.Init('CHASSIS','LTF_OP','OUT0201','a74',NVL_Outputs_States_CHASSIS.All.OUT0201,NVL_IO_CHASSIS.All_Outputs_Diag.OUT0201,Machine_IO.Node_CHASSIS);
Machine_IO.Outputs.LTR_OP.Init('CHASSIS','LTR_OP','OUT0202','a75',NVL_Outputs_States_CHASSIS.All.OUT0202,NVL_IO_CHASSIS.All_Outputs_Diag.OUT0202,Machine_IO.Node_CHASSIS);
Machine_IO.Outputs.RIGHTTRACKDIVERT_OP.Init('CHASSIS','RIGHTTRACKDIVERT_OP','OUT0203','a76',NVL_Outputs_States_CHASSIS.All.OUT0203,NVL_IO_CHASSIS.All_Outputs_Diag.OUT0203,Machine_IO.Node_CHASSIS);
Machine_IO.Outputs.RTF_OP.Init('CHASSIS','RTF_OP','OUT0204','a77',NVL_Outputs_States_CHASSIS.All.OUT0204,NVL_IO_CHASSIS.All_Outputs_Diag.OUT0204,Machine_IO.Node_CHASSIS);
Machine_IO.Outputs.RTR_OP.Init('CHASSIS','RTR_OP','OUT0205','a78',NVL_Outputs_States_CHASSIS.All.OUT0205,NVL_IO_CHASSIS.All_Outputs_Diag.OUT0205,Machine_IO.Node_CHASSIS);
Machine_IO.Outputs.DRUMONOFF_OP.Init('CHASSIS','DRUMONOFF_OP','OUT0206','a79',NVL_Outputs_States_CHASSIS.All.OUT0206,NVL_IO_CHASSIS.All_Outputs_Diag.OUT0206,Machine_IO.Node_CHASSIS);
Machine_IO.Outputs.FEEDERONOFF_OP.Init('CHASSIS','FEEDERONOFF_OP','OUT0207','a80',NVL_Outputs_States_CHASSIS.All.OUT0207,NVL_IO_CHASSIS.All_Outputs_Diag.OUT0207,Machine_IO.Node_CHASSIS);
Machine_IO.Outputs.ECUENABLE.Init('CHASSIS','ECUENABLE','OUT0208','a81',NVL_Outputs_States_CHASSIS.All.OUT0208,NVL_IO_CHASSIS.All_Outputs_Diag.OUT0208,Machine_IO.Node_CHASSIS);
Machine_IO.Outputs.SPARE_OUT3000.Init('CHASSIS','SPARE_OUT3000','OUT3000','a31',NVL_Outputs_States_CHASSIS.All.OUT3000,NVL_IO_CHASSIS.All_Outputs_Diag.OUT3000,Machine_IO.Node_CHASSIS);
Machine_IO.Outputs.SPARE_OUT3001.Init('CHASSIS','SPARE_OUT3001','OUT3001','a32',NVL_Outputs_States_CHASSIS.All.OUT3001,NVL_IO_CHASSIS.All_Outputs_Diag.OUT3001,Machine_IO.Node_CHASSIS);

// Machine_Link_Outputs_Init_CODE_GEN_STOP

END_PROGRAM

// App_CODE_GEN/MAIN_CODE_GEN/App_CODE_GEN/Machine IO/Funcs/Machine_Scale_Inputs
PROGRAM Machine_Scale_Inputs
VAR CONSTANT
END_VAR

VAR

END_VAR

END_PROGRAM

(* text list AlarmGroup_App (id | default | ge | en)
  101 | Emergencey Stop Active | Emergencey Stop Active | Emergencey Stop Active
  102 | PLC Ethernet Common Failure | PLC Ethernet Common Failure | PLC Ethernet Common Failure
  1100 | Ethernet - CHASSIS PLC Missing on powerup | Ethernet - CHASSIS PLC Missing on powerup | Ethernet - CHASSIS PLC Missing on powerup
  1101 | Ethernet - CHASSIS PLC - heartbeat less than error | Ethernet - CHASSIS PLC - heartbeat less than error | Ethernet - CHASSIS PLC - heartbeat less than error
  1102 | Ethernet - CHASSIS PLC - heartbeat difference error | Ethernet - CHASSIS PLC - heartbeat difference error | Ethernet - CHASSIS PLC - heartbeat difference error
  1103 | Ethernet - CHASSIS PLC - heartbeat frozen error | Ethernet - CHASSIS PLC - heartbeat frozen error | Ethernet - CHASSIS PLC - heartbeat frozen error
  1104 | Ethernet - CHASSIS PLC - heartbeat difference warning | Ethernet - CHASSIS PLC - heartbeat difference warning | Ethernet - CHASSIS PLC - heartbeat difference warning
  1105 | Ethernet - CHASSIS PLC - heartbeat frozen warning | Ethernet - CHASSIS PLC - heartbeat frozen warning | Ethernet - CHASSIS PLC - heartbeat frozen warning
  103 | Battery Voltage Warning | Battery Voltage Warning | Battery Voltage Warning
  104 | Hydraulic Oil level Low | Hydraulic Oil level Low | Hydraulic Oil level Low
   |  |  |  *)

(* text list AlarmGroup_IO (id | default | ge | en)
  1001 | ESTOPS_SAFETY_RELAY (CHASSIS.IN0100) | ESTOPS_SAFETY_RELAY (CHASSIS.IN0100) | ESTOPS_SAFETY_RELAY (CHASSIS.IN0100)
  1002 | OVERRIDE_GENERAL_SWT (CHASSIS.IN0101) | OVERRIDE_GENERAL_SWT (CHASSIS.IN0101) | OVERRIDE_GENERAL_SWT (CHASSIS.IN0101)
  1003 | FUNCTIONS_DEADMAN_CHASSIS_BTN (CHASSIS.IN0102) | FUNCTIONS_DEADMAN_CHASSIS_BTN (CHASSIS.IN0102) | FUNCTIONS_DEADMAN_CHASSIS_BTN (CHASSIS.IN0102)
  1004 | CABIN_RAISE_CHASSIS_BTN (CHASSIS.IN0103) | CABIN_RAISE_CHASSIS_BTN (CHASSIS.IN0103) | CABIN_RAISE_CHASSIS_BTN (CHASSIS.IN0103)
  1005 | CABIN_LOWER_CHASSIS_BTN (CHASSIS.IN0200) | CABIN_LOWER_CHASSIS_BTN (CHASSIS.IN0200) | CABIN_LOWER_CHASSIS_BTN (CHASSIS.IN0200)
  1006 | JACKLEGS_DOWN_CHASSIS_BTN (CHASSIS.IN0201) | JACKLEGS_DOWN_CHASSIS_BTN (CHASSIS.IN0201) | JACKLEGS_DOWN_CHASSIS_BTN (CHASSIS.IN0201)
  1007 | JACKLEGS_UP_CHASSIS_BTN (CHASSIS.IN0202) | JACKLEGS_UP_CHASSIS_BTN (CHASSIS.IN0202) | JACKLEGS_UP_CHASSIS_BTN (CHASSIS.IN0202)
  1008 | ENGINE_START_CHASSIS_BTN (CHASSIS.IN0203) | ENGINE_START_CHASSIS_BTN (CHASSIS.IN0203) | ENGINE_START_CHASSIS_BTN (CHASSIS.IN0203)
  1009 | HYDRAULICS_DC_PUMP_RUNNING_SIG (CHASSIS.IN0600) | HYDRAULICS_DC_PUMP_RUNNING_SIG (CHASSIS.IN0600) | HYDRAULICS_DC_PUMP_RUNNING_SIG (CHASSIS.IN0600)
  1010 | JACKLEGS_STOWED_DOWN_PRESSURE_SWT (CHASSIS.IN0601) | JACKLEGS_STOWED_DOWN_PRESSURE_SWT (CHASSIS.IN0601) | JACKLEGS_STOWED_DOWN_PRESSURE_SWT (CHASSIS.IN0601)
  1011 | JACKLEGS_STOWED_UP_PRESSURE_SWT (CHASSIS.IN0602) | JACKLEGS_STOWED_UP_PRESSURE_SWT (CHASSIS.IN0602) | JACKLEGS_STOWED_UP_PRESSURE_SWT (CHASSIS.IN0602)
  1012 | MAINS_AC_MAINS_CONNECTED (CHASSIS.IN0603) | MAINS_AC_MAINS_CONNECTED (CHASSIS.IN0603) | MAINS_AC_MAINS_CONNECTED (CHASSIS.IN0603)
  1013 | TRUCK_NEUTRAL_FROM_TRUCK  (CHASSIS.IN0700) | TRUCK_NEUTRAL_FROM_TRUCK  (CHASSIS.IN0700) | TRUCK_NEUTRAL_FROM_TRUCK  (CHASSIS.IN0700)
  1014 | SPARE_CHASSIS_IN0701 (CHASSIS.IN0701) | SPARE_CHASSIS_IN0701 (CHASSIS.IN0701) | SPARE_CHASSIS_IN0701 (CHASSIS.IN0701)
  1015 | CABIN_PART_RAISED_DIG (CHASSIS.IN0702) | CABIN_PART_RAISED_DIG (CHASSIS.IN0702) | CABIN_PART_RAISED_DIG (CHASSIS.IN0702)
  1016 | SPARE_CHASSIS_IN0703 (CHASSIS.IN0703) | SPARE_CHASSIS_IN0703 (CHASSIS.IN0703) | SPARE_CHASSIS_IN0703 (CHASSIS.IN0703)
  1017 | CABIN_LOWER_LIMIT_DIG (CHASSIS.IN0000) | CABIN_LOWER_LIMIT_DIG (CHASSIS.IN0000) | CABIN_LOWER_LIMIT_DIG (CHASSIS.IN0000)
  1018 | CABIN_FULLY_STOWED_DIG (CHASSIS.IN0001) | CABIN_FULLY_STOWED_DIG (CHASSIS.IN0001) | CABIN_FULLY_STOWED_DIG (CHASSIS.IN0001)
  1019 | PTO_ACTIVE_SIG (CHASSIS.IN0002) | PTO_ACTIVE_SIG (CHASSIS.IN0002) | PTO_ACTIVE_SIG (CHASSIS.IN0002)
  1020 | FUNCTIONS_CHASSIS_CABIN_CHANGE_OVER_SWT (CHASSIS.IN0003) | FUNCTIONS_CHASSIS_CABIN_CHANGE_OVER_SWT (CHASSIS.IN0003) | FUNCTIONS_CHASSIS_CABIN_CHANGE_OVER_SWT (CHASSIS.IN0003)
  1021 | LIGHTS_SIDE_LIGHTS_DASH_SIG (CHASSIS.IN0500) | LIGHTS_SIDE_LIGHTS_DASH_SIG (CHASSIS.IN0500) | LIGHTS_SIDE_LIGHTS_DASH_SIG (CHASSIS.IN0500)
  1022 | TRUCK_HANDBRAKE_APPLIED_SIGNAL (CHASSIS.IN0501) | TRUCK_HANDBRAKE_APPLIED_SIGNAL (CHASSIS.IN0501) | TRUCK_HANDBRAKE_APPLIED_SIGNAL (CHASSIS.IN0501)
  1023 | ENGINE_RUNNING_SIGNAL (CHASSIS.IN0502) | ENGINE_RUNNING_SIGNAL (CHASSIS.IN0502) | ENGINE_RUNNING_SIGNAL (CHASSIS.IN0502)
  1024 | TRUCK_REVERSE_FROM_TRUCK (CHASSIS.IN0503) | TRUCK_REVERSE_FROM_TRUCK (CHASSIS.IN0503) | TRUCK_REVERSE_FROM_TRUCK (CHASSIS.IN0503)
  1025 | SPARE_CHASSIS_IN0400 (CHASSIS.IN0400) | SPARE_CHASSIS_IN0400 (CHASSIS.IN0400) | SPARE_CHASSIS_IN0400 (CHASSIS.IN0400)
  1026 | ENGINE_STOP_CHASSIS_BTN (CHASSIS.IN0401) | ENGINE_STOP_CHASSIS_BTN (CHASSIS.IN0401) | ENGINE_STOP_CHASSIS_BTN (CHASSIS.IN0401)
  1027 | HYDRAULICS_OIL_LEVEL_RES (CHASSIS.IN0900) | HYDRAULICS_OIL_LEVEL_RES (CHASSIS.IN0900) | HYDRAULICS_OIL_LEVEL_RES (CHASSIS.IN0900)
  1028 | SPARE_CHASSIS_IN0901 (CHASSIS.IN0901) | SPARE_CHASSIS_IN0901 (CHASSIS.IN0901) | SPARE_CHASSIS_IN0901 (CHASSIS.IN0901)
  1029 | SPARE_CHASSIS_IN0300 (CHASSIS.IN0300) | SPARE_CHASSIS_IN0300 (CHASSIS.IN0300) | SPARE_CHASSIS_IN0300 (CHASSIS.IN0300)
  1030 | SPARE_CHASSIS_IN0301 (CHASSIS.IN0301) | SPARE_CHASSIS_IN0301 (CHASSIS.IN0301) | SPARE_CHASSIS_IN0301 (CHASSIS.IN0301)
  1031 | JACKLEGS_CYCLINDER_100_BAR_PRESSURE_SWT (CHASSIS.IN0800) | JACKLEGS_CYCLINDER_100_BAR_PRESSURE_SWT (CHASSIS.IN0800) | JACKLEGS_CYCLINDER_100_BAR_PRESSURE_SWT (CHASSIS.IN0800)
  1032 | JACKLEGS_CYCLINDER_150_BAR_PRESSURE_SWT (CHASSIS.IN0801) | JACKLEGS_CYCLINDER_150_BAR_PRESSURE_SWT (CHASSIS.IN0801) | JACKLEGS_CYCLINDER_150_BAR_PRESSURE_SWT (CHASSIS.IN0801)
  1033 | ENGINE_STOP_COMMAND (CHASSIS.OUT0000) | ENGINE_STOP_COMMAND (CHASSIS.OUT0000) | ENGINE_STOP_COMMAND (CHASSIS.OUT0000)
  1034 | CHASSIS_SIREN (CHASSIS.OUT0001) | CHASSIS_SIREN (CHASSIS.OUT0001) | CHASSIS_SIREN (CHASSIS.OUT0001)
  1035 | SPARE_CHASSIS_OUT0002 (CHASSIS.OUT0002) | SPARE_CHASSIS_OUT0002 (CHASSIS.OUT0002) | SPARE_CHASSIS_OUT0002 (CHASSIS.OUT0002)
  1036 | JACKLEGS_WARNING_BEACON (CHASSIS.OUT0003) | JACKLEGS_WARNING_BEACON (CHASSIS.OUT0003) | JACKLEGS_WARNING_BEACON (CHASSIS.OUT0003)
  1037 | HYDRAULICS_OIL_LEVEL_WARNING_LED (CHASSIS.OUT0004) | HYDRAULICS_OIL_LEVEL_WARNING_LED (CHASSIS.OUT0004) | HYDRAULICS_OIL_LEVEL_WARNING_LED (CHASSIS.OUT0004)
  1038 | SPARE_CHASSIS_OUT0005 (CHASSIS.OUT0005) | SPARE_CHASSIS_OUT0005 (CHASSIS.OUT0005) | SPARE_CHASSIS_OUT0005 (CHASSIS.OUT0005)
  1039 | HYDRAULICS_MASTER_VALVE (CHASSIS.OUT0006) | HYDRAULICS_MASTER_VALVE (CHASSIS.OUT0006) | HYDRAULICS_MASTER_VALVE (CHASSIS.OUT0006)
  1040 | PTO_TOGGLE (CHASSIS.OUT0007) | PTO_TOGGLE (CHASSIS.OUT0007) | PTO_TOGGLE (CHASSIS.OUT0007)
  1041 | SPARE_CHASSIS_OUT0008 (CHASSIS.OUT0008) | SPARE_CHASSIS_OUT0008 (CHASSIS.OUT0008) | SPARE_CHASSIS_OUT0008 (CHASSIS.OUT0008)
  1042 | CHASSIS_Supply_GROUP0 (CHASSIS.GROUP0) | CHASSIS_Supply_GROUP0 (CHASSIS.GROUP0) | CHASSIS_Supply_GROUP0 (CHASSIS.GROUP0)
  1043 | SPARE_CHASSIS_OUT0100 (CHASSIS.OUT0100) | SPARE_CHASSIS_OUT0100 (CHASSIS.OUT0100) | SPARE_CHASSIS_OUT0100 (CHASSIS.OUT0100)
  1044 | ENGINE_START_COMMAND (CHASSIS.OUT0101) | ENGINE_START_COMMAND (CHASSIS.OUT0101) | ENGINE_START_COMMAND (CHASSIS.OUT0101)
  1045 | SPARE_CHASSIS_OUT0102 (CHASSIS.OUT0102) | SPARE_CHASSIS_OUT0102 (CHASSIS.OUT0102) | SPARE_CHASSIS_OUT0102 (CHASSIS.OUT0102)
  1046 | PLATFORM_TRAVERSE_LEFT_VALVE (CHASSIS.OUT0103) | PLATFORM_TRAVERSE_LEFT_VALVE (CHASSIS.OUT0103) | PLATFORM_TRAVERSE_LEFT_VALVE (CHASSIS.OUT0103)
  1047 | SPARE_CHASSIS_OUT0104 (CHASSIS.OUT0104) | SPARE_CHASSIS_OUT0104 (CHASSIS.OUT0104) | SPARE_CHASSIS_OUT0104 (CHASSIS.OUT0104)
  1048 | CABIN_RAISE_COMMAND (CHASSIS.OUT0105) | CABIN_RAISE_COMMAND (CHASSIS.OUT0105) | CABIN_RAISE_COMMAND (CHASSIS.OUT0105)
  1049 | CABIN_LOWER_COMMAND (CHASSIS.OUT0106) | CABIN_LOWER_COMMAND (CHASSIS.OUT0106) | CABIN_LOWER_COMMAND (CHASSIS.OUT0106)
  1050 | JACKLEGS_UP_COMMAND (CHASSIS.OUT0107) | JACKLEGS_UP_COMMAND (CHASSIS.OUT0107) | JACKLEGS_UP_COMMAND (CHASSIS.OUT0107)
  1051 | JACKLEGS_DOWN_COMMAND (CHASSIS.OUT0108) | JACKLEGS_DOWN_COMMAND (CHASSIS.OUT0108) | JACKLEGS_DOWN_COMMAND (CHASSIS.OUT0108)
  1052 | CHASSIS_Supply_GROUP1 (CHASSIS.GROUP1) | CHASSIS_Supply_GROUP1 (CHASSIS.GROUP1) | CHASSIS_Supply_GROUP1 (CHASSIS.GROUP1)
  1053 | HYDRAULICS_MASTER_LED_CAB (CHASSIS.OUT0200) | HYDRAULICS_MASTER_LED_CAB (CHASSIS.OUT0200) | HYDRAULICS_MASTER_LED_CAB (CHASSIS.OUT0200)
  1054 | OVERRIDE_DRIVE_INTERLOCK_ACTIVE_LED (CHASSIS.OUT0201) | OVERRIDE_DRIVE_INTERLOCK_ACTIVE_LED (CHASSIS.OUT0201) | OVERRIDE_DRIVE_INTERLOCK_ACTIVE_LED (CHASSIS.OUT0201)
  1055 | CABIN_FULLY_STOWED_LED (CHASSIS.OUT0202) | CABIN_FULLY_STOWED_LED (CHASSIS.OUT0202) | CABIN_FULLY_STOWED_LED (CHASSIS.OUT0202)
  1056 | JACKLEGS_STOWED_LED (CHASSIS.OUT0203) | JACKLEGS_STOWED_LED (CHASSIS.OUT0203) | JACKLEGS_STOWED_LED (CHASSIS.OUT0203)
  1057 | JACKLEGS_DOWN_LED (CHASSIS.OUT0204) | JACKLEGS_DOWN_LED (CHASSIS.OUT0204) | JACKLEGS_DOWN_LED (CHASSIS.OUT0204)
  1058 | CABIN_RAISED_LED (CHASSIS.OUT0205) | CABIN_RAISED_LED (CHASSIS.OUT0205) | CABIN_RAISED_LED (CHASSIS.OUT0205)
  1059 | PLATFORM_TRAVERSE_RIGHT_VALVE (CHASSIS.OUT0206) | PLATFORM_TRAVERSE_RIGHT_VALVE (CHASSIS.OUT0206) | PLATFORM_TRAVERSE_RIGHT_VALVE (CHASSIS.OUT0206)
  1060 | PLATFORM_RETRACT_COMMAND (CHASSIS.OUT0207) | PLATFORM_RETRACT_COMMAND (CHASSIS.OUT0207) | PLATFORM_RETRACT_COMMAND (CHASSIS.OUT0207)
  1061 | PLATFORM_EXTEND_COMMAND (CHASSIS.OUT0208) | PLATFORM_EXTEND_COMMAND (CHASSIS.OUT0208) | PLATFORM_EXTEND_COMMAND (CHASSIS.OUT0208)
  1062 | CHASSIS_Supply_GROUP2 (CHASSIS.GROUP2) | CHASSIS_Supply_GROUP2 (CHASSIS.GROUP2) | CHASSIS_Supply_GROUP2 (CHASSIS.GROUP2)
  1063 | SPARE_CHASSIS_OUT3000 (CHASSIS.OUT3000) | SPARE_CHASSIS_OUT3000 (CHASSIS.OUT3000) | SPARE_CHASSIS_OUT3000 (CHASSIS.OUT3000)
  1064 | SPARE_CHASSIS_OUT3001 (CHASSIS.OUT3001) | SPARE_CHASSIS_OUT3001 (CHASSIS.OUT3001) | SPARE_CHASSIS_OUT3001 (CHASSIS.OUT3001)
  1200 | SPARE_CABIN_IN0100 (CABIN.IN0100) | SPARE_CABIN_IN0100 (CABIN.IN0100) | SPARE_CABIN_IN0100 (CABIN.IN0100)
  1201 | PLATFORM_EXTEND_BTN (CABIN.IN0101) | PLATFORM_EXTEND_BTN (CABIN.IN0101) | PLATFORM_EXTEND_BTN (CABIN.IN0101)
  1202 | PLATFORM_RETRACT_BTN (CABIN.IN0102) | PLATFORM_RETRACT_BTN (CABIN.IN0102) | PLATFORM_RETRACT_BTN (CABIN.IN0102)
  1203 | PLATFORM_SIDERAILS_LHS_SIDERAILS_STOWED_DIG (CABIN.IN0103) | PLATFORM_SIDERAILS_LHS_SIDERAILS_STOWED_DIG (CABIN.IN0103) | PLATFORM_SIDERAILS_LHS_SIDERAILS_STOWED_DIG (CABIN.IN0103)
  1204 | PLATFORM_SIDERAILS_RHS_SIDERAILS_STOWED_DIG (CABIN.IN0200) | PLATFORM_SIDERAILS_RHS_SIDERAILS_STOWED_DIG (CABIN.IN0200) | PLATFORM_SIDERAILS_RHS_SIDERAILS_STOWED_DIG (CABIN.IN0200)
  1205 | PLATFORM_TRAVERSE_STOWED_DIG (CABIN.IN0201) | PLATFORM_TRAVERSE_STOWED_DIG (CABIN.IN0201) | PLATFORM_TRAVERSE_STOWED_DIG (CABIN.IN0201)
  1206 | SPARE_CABIN_IN0202 (CABIN.IN0202) | SPARE_CABIN_IN0202 (CABIN.IN0202) | SPARE_CABIN_IN0202 (CABIN.IN0202)
  1207 | PLATFORM_LEUZE_SENSORS_LEFT_SENSOR_DIG (CABIN.IN0203) | PLATFORM_LEUZE_SENSORS_LEFT_SENSOR_DIG (CABIN.IN0203) | PLATFORM_LEUZE_SENSORS_LEFT_SENSOR_DIG (CABIN.IN0203)
  1208 | PLATFORM_LEUZE_SENSORS_RIGHT_SENSOR_DIG (CABIN.IN0600) | PLATFORM_LEUZE_SENSORS_RIGHT_SENSOR_DIG (CABIN.IN0600) | PLATFORM_LEUZE_SENSORS_RIGHT_SENSOR_DIG (CABIN.IN0600)
  1209 | PLATFORM_FULLY_STOWED_DIG (CABIN.IN0601) | PLATFORM_FULLY_STOWED_DIG (CABIN.IN0601) | PLATFORM_FULLY_STOWED_DIG (CABIN.IN0601)
  1210 | PLATFORM_PART_STOWED_DIG (CABIN.IN0602) | PLATFORM_PART_STOWED_DIG (CABIN.IN0602) | PLATFORM_PART_STOWED_DIG (CABIN.IN0602)
  1211 | DOORS_REAR_DOOR_CLOSED_SIG (CABIN.IN0603) | DOORS_REAR_DOOR_CLOSED_SIG (CABIN.IN0603) | DOORS_REAR_DOOR_CLOSED_SIG (CABIN.IN0603)
  1212 | PLATFORM_SAFETY_GATES_LHS_EDGE_SENSOR (CABIN.IN0700) | PLATFORM_SAFETY_GATES_LHS_EDGE_SENSOR (CABIN.IN0700) | PLATFORM_SAFETY_GATES_LHS_EDGE_SENSOR (CABIN.IN0700)
  1213 | SPARE_CABIN_IN0701 (CABIN.IN0701) | SPARE_CABIN_IN0701 (CABIN.IN0701) | SPARE_CABIN_IN0701 (CABIN.IN0701)
  1214 | SPARE_CABIN_IN0702 (CABIN.IN0702) | SPARE_CABIN_IN0702 (CABIN.IN0702) | SPARE_CABIN_IN0702 (CABIN.IN0702)
  1215 | PLATFORM_SAFETY_GATES_RHS_EDGE_SENSOR (CABIN.IN0703) | PLATFORM_SAFETY_GATES_RHS_EDGE_SENSOR (CABIN.IN0703) | PLATFORM_SAFETY_GATES_RHS_EDGE_SENSOR (CABIN.IN0703)
  1216 | SPARE_CABIN_IN0000 (CABIN.IN0000) | SPARE_CABIN_IN0000 (CABIN.IN0000) | SPARE_CABIN_IN0000 (CABIN.IN0000)
  1217 | PLATFORM_SAFETY_GATES_LHS_GATE_CLOSED_SIGNAL (CABIN.IN0001) | PLATFORM_SAFETY_GATES_LHS_GATE_CLOSED_SIGNAL (CABIN.IN0001) | PLATFORM_SAFETY_GATES_LHS_GATE_CLOSED_SIGNAL (CABIN.IN0001)
  1218 | PLATFORM_SAFETY_GATES_RHS_GATE_CLOSED_SIGNAL (CABIN.IN0002) | PLATFORM_SAFETY_GATES_RHS_GATE_CLOSED_SIGNAL (CABIN.IN0002) | PLATFORM_SAFETY_GATES_RHS_GATE_CLOSED_SIGNAL (CABIN.IN0002)
  1219 | SPARE_CABIN_IN0003 (CABIN.IN0003) | SPARE_CABIN_IN0003 (CABIN.IN0003) | SPARE_CABIN_IN0003 (CABIN.IN0003)
  1220 | CAS_RESET_SWT (CABIN.IN0500) | CAS_RESET_SWT (CABIN.IN0500) | CAS_RESET_SWT (CABIN.IN0500)
  1221 | CAS_TORTOISE_SWT (CABIN.IN0501) | CAS_TORTOISE_SWT (CABIN.IN0501) | CAS_TORTOISE_SWT (CABIN.IN0501)
  1222 | CAS_ENABLE_ON_OFF_SWT (CABIN.IN0502) | CAS_ENABLE_ON_OFF_SWT (CABIN.IN0502) | CAS_ENABLE_ON_OFF_SWT (CABIN.IN0502)
  1223 | SPARE_CABIN_IN0503 (CABIN.IN0503) | SPARE_CABIN_IN0503 (CABIN.IN0503) | SPARE_CABIN_IN0503 (CABIN.IN0503)
  1224 | PLATFORM_SAFETY_EDGE_SAFETY_BUMPER_RES_ANA (CABIN.IN0400) | PLATFORM_SAFETY_EDGE_SAFETY_BUMPER_RES_ANA (CABIN.IN0400) | PLATFORM_SAFETY_EDGE_SAFETY_BUMPER_RES_ANA (CABIN.IN0400)
  1225 | SPARE_CABIN_IN0401 (CABIN.IN0401) | SPARE_CABIN_IN0401 (CABIN.IN0401) | SPARE_CABIN_IN0401 (CABIN.IN0401)
  1226 | PLATFORM_TRAVERSE_LEFT_BTN (CABIN.IN0900) | PLATFORM_TRAVERSE_LEFT_BTN (CABIN.IN0900) | PLATFORM_TRAVERSE_LEFT_BTN (CABIN.IN0900)
  1227 | PLATFORM_TRAVERSE_RIGHT_BTN (CABIN.IN0901) | PLATFORM_TRAVERSE_RIGHT_BTN (CABIN.IN0901) | PLATFORM_TRAVERSE_RIGHT_BTN (CABIN.IN0901)
  1228 | DOORS_SIDE_DOOR_CLOSED_SIG (CABIN.IN0300) | DOORS_SIDE_DOOR_CLOSED_SIG (CABIN.IN0300) | DOORS_SIDE_DOOR_CLOSED_SIG (CABIN.IN0300)
  1229 | FUNCTIONS_DEADMAN_CABIN_BTN (CABIN.IN0301) | FUNCTIONS_DEADMAN_CABIN_BTN (CABIN.IN0301) | FUNCTIONS_DEADMAN_CABIN_BTN (CABIN.IN0301)
  1230 | SPARE_CABIN_IN0800 (CABIN.IN0800) | SPARE_CABIN_IN0800 (CABIN.IN0800) | SPARE_CABIN_IN0800 (CABIN.IN0800)
  1231 | SPARE_CABIN_IN0801 (CABIN.IN0801) | SPARE_CABIN_IN0801 (CABIN.IN0801) | SPARE_CABIN_IN0801 (CABIN.IN0801)
  1232 | PLATFORM_SIDERAILS_SIDERAILS_STOWED_LED (CABIN.OUT0000) | PLATFORM_SIDERAILS_SIDERAILS_STOWED_LED (CABIN.OUT0000) | PLATFORM_SIDERAILS_SIDERAILS_STOWED_LED (CABIN.OUT0000)
  1233 | PLATFORM_SAFETY_GATES_UNLOCK_1 (CABIN.OUT0001) | PLATFORM_SAFETY_GATES_UNLOCK_1 (CABIN.OUT0001) | PLATFORM_SAFETY_GATES_UNLOCK_1 (CABIN.OUT0001)
  1234 | TRUCK_FORCE_NEUTRAL (CABIN.OUT0002) | TRUCK_FORCE_NEUTRAL (CABIN.OUT0002) | TRUCK_FORCE_NEUTRAL (CABIN.OUT0002)
  1235 | PLATFORM_SAFETY_GATES_UNLOCK_2 (CABIN.OUT0003) | PLATFORM_SAFETY_GATES_UNLOCK_2 (CABIN.OUT0003) | PLATFORM_SAFETY_GATES_UNLOCK_2 (CABIN.OUT0003)
  1236 | CAS_LOCKOUT_LED (CABIN.OUT0004) | CAS_LOCKOUT_LED (CABIN.OUT0004) | CAS_LOCKOUT_LED (CABIN.OUT0004)
  1237 | PLATFORM_EXTENDED_LED (CABIN.OUT0005) | PLATFORM_EXTENDED_LED (CABIN.OUT0005) | PLATFORM_EXTENDED_LED (CABIN.OUT0005)
  1238 | PLATFORM_RETRACTED_LED (CABIN.OUT0006) | PLATFORM_RETRACTED_LED (CABIN.OUT0006) | PLATFORM_RETRACTED_LED (CABIN.OUT0006)
  1239 | CAS_TORTOISE_MODE_LED (CABIN.OUT0007) | CAS_TORTOISE_MODE_LED (CABIN.OUT0007) | CAS_TORTOISE_MODE_LED (CABIN.OUT0007)
  1240 | CAS_DRIVERS_BUZZER (CABIN.OUT0008) | CAS_DRIVERS_BUZZER (CABIN.OUT0008) | CAS_DRIVERS_BUZZER (CABIN.OUT0008)
  1241 | CABIN_Supply_GROUP0 (CABIN.GROUP0) | CABIN_Supply_GROUP0 (CABIN.GROUP0) | CABIN_Supply_GROUP0 (CABIN.GROUP0)
  1242 | DOORS_ALLOW_SIDE_DOOR (CABIN.OUT0100) | DOORS_ALLOW_SIDE_DOOR (CABIN.OUT0100) | DOORS_ALLOW_SIDE_DOOR (CABIN.OUT0100)
  1243 | DOORS_ALLOW_REAR_DOOR (CABIN.OUT0101) | DOORS_ALLOW_REAR_DOOR (CABIN.OUT0101) | DOORS_ALLOW_REAR_DOOR (CABIN.OUT0101)
  1244 | SPARE_CABIN_OUT0102 (CABIN.OUT0102) | SPARE_CABIN_OUT0102 (CABIN.OUT0102) | SPARE_CABIN_OUT0102 (CABIN.OUT0102)
  1245 | SPARE_CABIN_OUT0103 (CABIN.OUT0103) | SPARE_CABIN_OUT0103 (CABIN.OUT0103) | SPARE_CABIN_OUT0103 (CABIN.OUT0103)
  1246 | SPARE_CABIN_OUT0104 (CABIN.OUT0104) | SPARE_CABIN_OUT0104 (CABIN.OUT0104) | SPARE_CABIN_OUT0104 (CABIN.OUT0104)
  1247 | SPARE_CABIN_OUT0105 (CABIN.OUT0105) | SPARE_CABIN_OUT0105 (CABIN.OUT0105) | SPARE_CABIN_OUT0105 (CABIN.OUT0105)
  1248 | SPARE_CABIN_OUT0106 (CABIN.OUT0106) | SPARE_CABIN_OUT0106 (CABIN.OUT0106) | SPARE_CABIN_OUT0106 (CABIN.OUT0106)
  1249 | SPARE_CABIN_OUT0107 (CABIN.OUT0107) | SPARE_CABIN_OUT0107 (CABIN.OUT0107) | SPARE_CABIN_OUT0107 (CABIN.OUT0107)
  1250 | SPARE_CABIN_OUT0108 (CABIN.OUT0108) | SPARE_CABIN_OUT0108 (CABIN.OUT0108) | SPARE_CABIN_OUT0108 (CABIN.OUT0108)
  1251 | CABIN_Supply_GROUP1 (CABIN.GROUP1) | CABIN_Supply_GROUP1 (CABIN.GROUP1) | CABIN_Supply_GROUP1 (CABIN.GROUP1)
  1252 | SPARE_CABIN_OUT0200 (CABIN.OUT0200) | SPARE_CABIN_OUT0200 (CABIN.OUT0200) | SPARE_CABIN_OUT0200 (CABIN.OUT0200)
  1253 | LIGHTS_LEFT_SIDE_LIGHTS (CABIN.OUT0201) | LIGHTS_LEFT_SIDE_LIGHTS (CABIN.OUT0201) | LIGHTS_LEFT_SIDE_LIGHTS (CABIN.OUT0201)
  1254 | CAS_GREEN_BEACON (CABIN.OUT0202) | CAS_GREEN_BEACON (CABIN.OUT0202) | CAS_GREEN_BEACON (CABIN.OUT0202)
  1255 | FUNCTIONS_DEADMAN_CABIN_BTN_LED (CABIN.OUT0203) | FUNCTIONS_DEADMAN_CABIN_BTN_LED (CABIN.OUT0203) | FUNCTIONS_DEADMAN_CABIN_BTN_LED (CABIN.OUT0203)
  1256 | SPARE_CABIN_OUT0204 (CABIN.OUT0204) | SPARE_CABIN_OUT0204 (CABIN.OUT0204) | SPARE_CABIN_OUT0204 (CABIN.OUT0204)
  1257 | SPARE_CABIN_OUT0205 (CABIN.OUT0205) | SPARE_CABIN_OUT0205 (CABIN.OUT0205) | SPARE_CABIN_OUT0205 (CABIN.OUT0205)
  1258 | LIGHTS_SIDE_RLY (CABIN.OUT0206) | LIGHTS_SIDE_RLY (CABIN.OUT0206) | LIGHTS_SIDE_RLY (CABIN.OUT0206)
  1259 | SPARE_CABIN_OUT0207 (CABIN.OUT0207) | SPARE_CABIN_OUT0207 (CABIN.OUT0207) | SPARE_CABIN_OUT0207 (CABIN.OUT0207)
  1260 | SPARE_CABIN_OUT0208 (CABIN.OUT0208) | SPARE_CABIN_OUT0208 (CABIN.OUT0208) | SPARE_CABIN_OUT0208 (CABIN.OUT0208)
  1261 | CABIN_Supply_GROUP2 (CABIN.GROUP2) | CABIN_Supply_GROUP2 (CABIN.GROUP2) | CABIN_Supply_GROUP2 (CABIN.GROUP2)
  1262 | SPARE_CABIN_OUT3000 (CABIN.OUT3000) | SPARE_CABIN_OUT3000 (CABIN.OUT3000) | SPARE_CABIN_OUT3000 (CABIN.OUT3000)
  1263 | SPARE_CABIN_OUT3001 (CABIN.OUT3001) | SPARE_CABIN_OUT3001 (CABIN.OUT3001) | SPARE_CABIN_OUT3001 (CABIN.OUT3001)
   |  |  |  *)

(* text list TextList_IO_Diag (id | default)
  CHASSIS.IN0100 | ESTOP_OK
  CHASSIS.IN0101 | DRUM_PRESSURE
  CHASSIS.IN0102 | SPARE_IN0102
  CHASSIS.IN0103 | SPARE_IN0103
  CHASSIS.IN0200 | SPARE_IN0200
  CHASSIS.IN0201 | SPARE_IN0201
  CHASSIS.IN0202 | SPARE_IN0202
  CHASSIS.IN0203 | SPARE_IN0203
  CHASSIS.IN0600 | SPARE_IN0600
  CHASSIS.IN0601 | SPARE_IN0601
  CHASSIS.IN0602 | JACKLEGS_STOWED_UP_PRESSURE_SWT
  CHASSIS.IN0603 | MAINS_AC_MAINS_CONNECTED
  CHASSIS.IN0700 | TRUCK_NEUTRAL_FROM_TRUCK 
  CHASSIS.IN0701 | SPARE_CHASSIS_IN0701
  CHASSIS.IN0702 | CABIN_PART_RAISED_DIG
  CHASSIS.IN0703 | SPARE_CHASSIS_IN0703
  CHASSIS.IN0000 | CABIN_LOWER_LIMIT_DIG
  CHASSIS.IN0001 | CABIN_FULLY_STOWED_DIG
  CHASSIS.IN0002 | PTO_ACTIVE_SIG
  CHASSIS.IN0003 | FUNCTIONS_CHASSIS_CABIN_CHANGE_OVER_SWT
  CHASSIS.IN0500 | LIGHTS_SIDE_LIGHTS_DASH_SIG
  CHASSIS.IN0501 | TRUCK_HANDBRAKE_APPLIED_SIGNAL
  CHASSIS.IN0502 | ENGINE_RUNNING_SIGNAL
  CHASSIS.IN0503 | TRUCK_REVERSE_FROM_TRUCK
  CHASSIS.IN0400 | SPARE_CHASSIS_IN0400
  CHASSIS.IN0401 | ENGINE_STOP_CHASSIS_BTN
  CHASSIS.IN0900 | HYDRAULICS_OIL_LEVEL_RES
  CHASSIS.IN0901 | SPARE_CHASSIS_IN0901
  CHASSIS.IN0300 | SPARE_CHASSIS_IN0300
  CHASSIS.IN0301 | SPARE_CHASSIS_IN0301
  CHASSIS.IN0800 | JACKLEGS_CYCLINDER_100_BAR_PRESSURE_SWT
  CHASSIS.IN0801 | JACKLEGS_CYCLINDER_150_BAR_PRESSURE_SWT
  CHASSIS.OUT0000 | ENGINE_STOP_COMMAND
  CHASSIS.OUT0001 | CHASSIS_SIREN
  CHASSIS.OUT0002 | SPARE_CHASSIS_OUT0002
  CHASSIS.OUT0003 | JACKLEGS_WARNING_BEACON
  CHASSIS.OUT0004 | HYDRAULICS_OIL_LEVEL_WARNING_LED
  CHASSIS.OUT0005 | SPARE_CHASSIS_OUT0005
  CHASSIS.OUT0006 | HYDRAULICS_MASTER_VALVE
  CHASSIS.OUT0007 | PTO_TOGGLE
  CHASSIS.OUT0008 | SPARE_CHASSIS_OUT0008
  CHASSIS.GROUP0 | CHASSIS_Supply_GROUP0
  CHASSIS.OUT0100 | SPARE_CHASSIS_OUT0100
  CHASSIS.OUT0101 | ENGINE_START_COMMAND
  CHASSIS.OUT0102 | SPARE_CHASSIS_OUT0102
  CHASSIS.OUT0103 | PLATFORM_TRAVERSE_LEFT_VALVE
  CHASSIS.OUT0104 | SPARE_CHASSIS_OUT0104
  CHASSIS.OUT0105 | CABIN_RAISE_COMMAND
  CHASSIS.OUT0106 | CABIN_LOWER_COMMAND
  CHASSIS.OUT0107 | JACKLEGS_UP_COMMAND
  CHASSIS.OUT0108 | JACKLEGS_DOWN_COMMAND
  CHASSIS.GROUP1 | CHASSIS_Supply_GROUP1
  CHASSIS.OUT0200 | HYDRAULICS_MASTER_LED_CAB
  CHASSIS.OUT0201 | OVERRIDE_DRIVE_INTERLOCK_ACTIVE_LED
  CHASSIS.OUT0202 | CABIN_FULLY_STOWED_LED
  CHASSIS.OUT0203 | JACKLEGS_STOWED_LED
  CHASSIS.OUT0204 | JACKLEGS_DOWN_LED
  CHASSIS.OUT0205 | CABIN_RAISED_LED
  CHASSIS.OUT0206 | PLATFORM_TRAVERSE_RIGHT_VALVE
  CHASSIS.OUT0207 | PLATFORM_RETRACT_COMMAND
  CHASSIS.OUT0208 | PLATFORM_EXTEND_COMMAND
  CHASSIS.GROUP2 | CHASSIS_Supply_GROUP2
  CHASSIS.OUT3000 | SPARE_CHASSIS_OUT3000
  CHASSIS.OUT3001 | SPARE_CHASSIS_OUT3001
   |  *)
